(* CODESYS project TripleDoor.project

Project tree, tasks and I/O mapping:
  Device : CODESYS Control Win V3 x64, 3S - Smart Software Solutions GmbH, version 3.5.11.0
    application Application
      libraries: Standard, * (System); VisuDialogs, * (System); Util, * (System)
      task MainTask (cyclic, interval t#10ms, priority 1) calls Plant, Controller
      program Plant [ST]
      visualisation Visualization
      global variables GVL
      program Controller [ST]
  text list GlobalTextList
*)

// Device/Application/GVL
{attribute 'qualified_only' := 'false'}
VAR_GLOBAL
    (* Presence sensors *)
    presenceSideA           : BOOL;
    presenceSideB           : BOOL;
    (* Presence triggers - visualization writes here *)
    presenceTriggerA        : BOOL;
    presenceTriggerB        : BOOL;
    (* Partition pressure sensor *)
    partitionPressure       : BOOL;
    (* Manual rotation buttons *)
    rotateForwardButton     : BOOL;
    rotateBackwardButton    : BOOL;
    (* Rotation direction: FALSE=counter-clockwise (default), TRUE=clockwise *)
    rotationClockwise       : BOOL;
    (* Door angle sensor *)
    doorAngle               : REAL;
(* Rotation status *)
    isRotating              : BOOL;
    (* Motor control *)
    motorOn                 : BOOL;
    rotationForward         : BOOL;
    (* Motor enable switch *)
    motorEnable             : BOOL := TRUE;
    (* Emergency stop *)
    emergencyStop           : BOOL;
    (* Traffic lights *)
    lightSideA              : BOOL;
    lightSideB              : BOOL;
END_VAR

// Device/Application/Plant
PROGRAM Plant
VAR CONSTANT
    ROTATION_SPEED  : REAL := 0.1;
    MAX_ANGLE       : REAL := 360.0;
    PRESENCE_HOLD   : INT := 500;
END_VAR
VAR
    initialized      : BOOL := FALSE;
    presenceTimerA   : INT := 0;
    presenceTimerB   : INT := 0;
END_VAR

IF NOT initialized THEN
    GVL.doorAngle            := 0.0;
    GVL.presenceSideA        := FALSE;
    GVL.presenceSideB        := FALSE;
    GVL.presenceTriggerA     := FALSE;
    GVL.presenceTriggerB     := FALSE;
    presenceTimerA           := 0;
    presenceTimerB           := 0;
    initialized              := TRUE;
END_IF

(* Presence hold - trigger is set by visualization, timer keeps presence active *)
IF GVL.presenceTriggerA THEN
    presenceTimerA := PRESENCE_HOLD;
    GVL.presenceTriggerA := FALSE;
END_IF
GVL.presenceSideA := (presenceTimerA > 0);
IF presenceTimerA > 0 THEN
    presenceTimerA := presenceTimerA - 1;
END_IF

IF GVL.presenceTriggerB THEN
    presenceTimerB := PRESENCE_HOLD;
    GVL.presenceTriggerB := FALSE;
END_IF
GVL.presenceSideB := (presenceTimerB > 0);
IF presenceTimerB > 0 THEN
    presenceTimerB := presenceTimerB - 1;
END_IF

(* MotorSim *)
GVL.isRotating := GVL.motorOn;

(* DoorRotationSim *)
IF GVL.isRotating THEN
    IF GVL.rotationForward THEN
        GVL.doorAngle := GVL.doorAngle - ROTATION_SPEED;
    ELSE
        GVL.doorAngle := GVL.doorAngle + ROTATION_SPEED;
    END_IF
END_IF

IF GVL.doorAngle >= MAX_ANGLE THEN
    GVL.doorAngle := GVL.doorAngle - MAX_ANGLE;
END_IF
IF GVL.doorAngle < 0.0 THEN
    GVL.doorAngle := GVL.doorAngle + MAX_ANGLE;
END_IF

END_PROGRAM

// Device/Application/Controller
PROGRAM Controller
VAR CONSTANT
    ROTATION_TIME   : INT := 100;
    REVERSE_TICKS   : INT := 50;    (* 5 degrees at ROTATION_SPEED=0.1 *)
END_VAR
VAR
    (* MainControl state: 0=idle, 1=rotating, 2=manualRotation, 3=pressure *)
    mainState               : INT := 0;
    timer                   : INT := 0;
    manualActive            : BOOL := FALSE;
    manualDirectionForward  : BOOL := TRUE;
    (* Pressure sub-process: 0=released, 1=reversing, 2=stopped *)
    pauseState              : INT := 0;
    reverseCounter          : INT := 0;
END_VAR

(* Emergency stop - disable motor *)
IF GVL.emergencyStop THEN
    GVL.motorEnable := FALSE;
END_IF

(* Motor disabled - immediate stop, reset to idle *)
IF NOT GVL.motorEnable THEN
    GVL.motorOn := FALSE;
    GVL.rotationForward := NOT GVL.rotationClockwise;
    GVL.lightSideA := FALSE;
    GVL.lightSideB := FALSE;
	GVL.presenceSideA := FALSE;	
    GVL.presenceSideB := FALSE;
    manualActive := FALSE;
    timer := 0;
    pauseState := 0;
    mainState := 0;
ELSE

CASE mainState OF

0: (* idle *)
    GVL.lightSideA := TRUE;
    GVL.lightSideB := TRUE;
    IF GVL.rotateForwardButton AND NOT GVL.rotateBackwardButton AND NOT GVL.partitionPressure THEN
        manualActive := TRUE;
        manualDirectionForward := TRUE;
        GVL.motorOn := TRUE;
        GVL.rotationForward := NOT GVL.rotationClockwise;
        GVL.lightSideA := TRUE;
        GVL.lightSideB := TRUE;
        mainState := 2;

    ELSIF GVL.rotateBackwardButton AND NOT GVL.rotateForwardButton AND NOT GVL.partitionPressure THEN
        manualActive := TRUE;
        manualDirectionForward := FALSE;
        GVL.motorOn := TRUE;
        GVL.rotationForward := GVL.rotationClockwise;
        GVL.lightSideA := TRUE;
        GVL.lightSideB := TRUE;
        mainState := 2;

    ELSIF (GVL.presenceSideA OR GVL.presenceSideB) AND NOT GVL.partitionPressure THEN
        manualActive := FALSE;
        manualDirectionForward := TRUE;
        GVL.motorOn := TRUE;
        GVL.rotationForward := NOT GVL.rotationClockwise;
        GVL.lightSideA := TRUE;
        GVL.lightSideB := TRUE;
        timer := ROTATION_TIME;
        mainState := 1;
    END_IF

1: (* rotating *)
    IF (GVL.presenceSideA OR GVL.presenceSideB) THEN
        timer := ROTATION_TIME;
    END_IF

    IF GVL.partitionPressure THEN
        GVL.motorOn := FALSE;
        GVL.rotationForward := NOT GVL.rotationForward;
        GVL.lightSideA := FALSE;
        GVL.lightSideB := FALSE;
        reverseCounter := REVERSE_TICKS;
        pauseState := 1;
        mainState := 3;
    END_IF

    IF mainState = 1 THEN
        timer := timer - 1;
    END_IF
    IF timer <= 0 AND mainState = 1 THEN
        GVL.motorOn := FALSE;
        GVL.rotationForward := NOT GVL.rotationClockwise;
        GVL.lightSideA := TRUE;
        GVL.lightSideB := TRUE;
        mainState := 0;
    END_IF

2: (* manualRotation *)
    IF GVL.partitionPressure THEN
        GVL.motorOn := FALSE;
        GVL.rotationForward := NOT GVL.rotationForward;
        GVL.lightSideA := FALSE;
        GVL.lightSideB := FALSE;
        reverseCounter := REVERSE_TICKS;
        pauseState := 1;
        mainState := 3;

    ELSIF GVL.rotateForwardButton AND GVL.rotateBackwardButton THEN
        GVL.motorOn := FALSE;
        GVL.rotationForward := NOT GVL.rotationClockwise;
        GVL.lightSideA := TRUE;
        GVL.lightSideB := TRUE;
        manualActive := FALSE;
        mainState := 0;

    ELSIF manualDirectionForward AND GVL.rotateForwardButton THEN
        GVL.motorOn := TRUE;
        GVL.rotationForward := NOT GVL.rotationClockwise;
        GVL.lightSideA := TRUE;
        GVL.lightSideB := TRUE;

    ELSIF (NOT manualDirectionForward) AND GVL.rotateBackwardButton THEN
        GVL.motorOn := TRUE;
        GVL.rotationForward := GVL.rotationClockwise;
        GVL.lightSideA := TRUE;
        GVL.lightSideB := TRUE;

    ELSE
        GVL.motorOn := FALSE;
        GVL.rotationForward := NOT GVL.rotationClockwise;
        GVL.lightSideA := TRUE;
        GVL.lightSideB := TRUE;
        manualActive := FALSE;
        mainState := 0;
    END_IF

3: (* pressure reaction *)
    IF pauseState = 1 THEN
        (* Reversing 5 degrees *)
        GVL.motorOn := TRUE;
        reverseCounter := reverseCounter - 1;
        IF reverseCounter <= 0 THEN
            GVL.motorOn := FALSE;
            pauseState := 2;
        END_IF
    END_IF

    IF pauseState = 2 THEN
        (* Stopped until pressure released *)
        GVL.motorOn := FALSE;
        IF NOT GVL.partitionPressure THEN
            pauseState := 0;
        END_IF
    END_IF

    IF pauseState = 0 THEN
        (* Pressure released - resume *)
        IF manualActive THEN
            IF manualDirectionForward AND GVL.rotateForwardButton THEN
                GVL.motorOn := TRUE;
                GVL.rotationForward := NOT GVL.rotationClockwise;
                GVL.lightSideA := TRUE;
                GVL.lightSideB := TRUE;
                mainState := 2;
            ELSIF (NOT manualDirectionForward) AND GVL.rotateBackwardButton THEN
                GVL.motorOn := TRUE;
                GVL.rotationForward := GVL.rotationClockwise;
                GVL.lightSideA := TRUE;
                GVL.lightSideB := TRUE;
                mainState := 2;
            ELSE
                GVL.motorOn := FALSE;
                GVL.rotationForward := NOT GVL.rotationClockwise;
                GVL.lightSideA := TRUE;
                GVL.lightSideB := TRUE;
                manualActive := FALSE;
                mainState := 0;
            END_IF
        ELSIF timer > 0 THEN
            GVL.motorOn := TRUE;
            GVL.rotationForward := NOT GVL.rotationClockwise;
            GVL.lightSideA := TRUE;
            GVL.lightSideB := TRUE;
            mainState := 1;
        ELSE
            GVL.motorOn := FALSE;
            GVL.rotationForward := NOT GVL.rotationClockwise;
            GVL.lightSideA := TRUE;
            GVL.lightSideB := TRUE;
            mainState := 0;
        END_IF
    END_IF

END_CASE

END_IF (* motorEnable / emergencyStop *)

END_PROGRAM

// Device/Application/Visualization
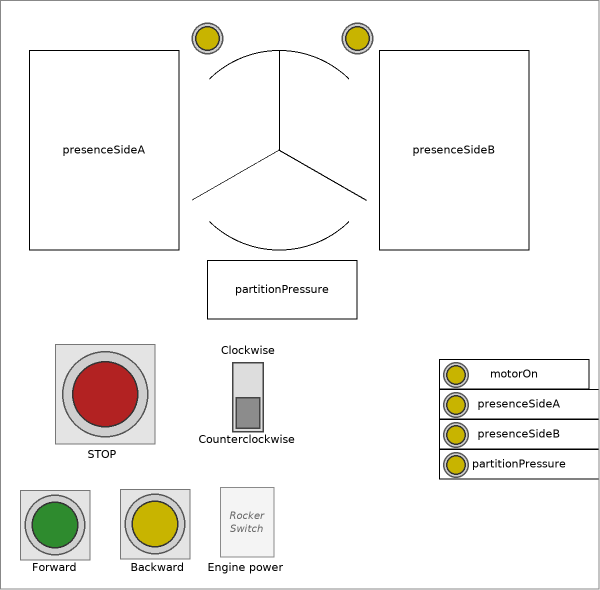
VISUALIZATION Visualization  // 600x590
    Rectangle (52,429 100x51), "STOP"
    Ellipse (179,50 200x200)
    Rectangle (59,50 150x200)
    Rectangle (349,50 150x200)
    RoundedRectangle (29,50 150x200), "presenceSideA"
        OnMouseMove: execute { GVL.presenceTriggerA := TRUE; }
        OnMouseEnter: execute { GVL.presenceTriggerA := TRUE; }
    RoundedRectangle (379,50 150x200), "presenceSideB"
        OnMouseMove: execute { GVL.presenceTriggerB := TRUE; }
        OnMouseEnter: execute { GVL.presenceTriggerB := TRUE; }
    PushSwitch (51,344 108x100), tooltip "Backward", variable: GVL.emergencyStop, behaviour: TAP, style: Switch-PushSwitch-Red
    Lamp1 (339,20 37x37), variable: GVL.lightSideB, style: Lamp-Lamp1-Yellow
    Lamp1 (189,20 37x37), variable: GVL.lightSideA, style: Lamp-Lamp1-Yellow
    Polyline (279,50) (279,150) (366,200) (279,150) (192,200)
        p2858320360: GVL.doorAngle
    Rectangle (207,260 150x59), "partitionPressure"
        OnMouseLeave: execute { GVL.partitionPressure := FALSE; }
        OnMouseEnter: execute { GVL.partitionPressure := TRUE; }
    Group (439,359 160x31)
        RoundedRectangle (0,0 150x30), "motorOn"
        Lamp1 (2,1 30x30), variable: GVL.motorOn, style: Lamp-Lamp1-Yellow
    RoundedRectangle (439,389 160x30), "presenceSideA"
    Lamp1 (441,390 30x30), variable: GVL.presenceSideA, style: Lamp-Lamp1-Yellow
    RoundedRectangle (439,419 160x30), "presenceSideB"
    Lamp1 (441,420 30x30), variable: GVL.presenceSideB, style: Lamp-Lamp1-Yellow
    RoundedRectangle (439,449 160x30), "partitionPressure"
    Lamp1 (441,450 30x30), variable: GVL.partitionPressure, style: Lamp-Lamp1-Yellow
    Rectangle (10,553 89x29), "Forward"
    Rectangle (113,553 89x29), "Backward"
    Rectangle (201,553 89x29), "Engine power"
    RockerSwitch (220,487 54x70), tooltip "Engine", variable: GVL.motorEnable, behaviour: TOGGLE, style: Switch-RockerSwitch-Red
    PushSwitch (120,489 70x70), tooltip "Backward", variable: GVL.rotateBackwardButton, behaviour: TAP, style: Switch-PushSwitch-Yellow
    PushSwitch (20,490 70x70), tooltip "Forward", variable: GVL.rotateForwardButton, behaviour: TAP, style: Switch-PushSwitch-Green
    Rectangle (192,425 110x29), "Counterclockwise"
    Rectangle (193,336 110x29), "Clockwise"
    DipSwitch (213,362 70x70), variable: GVL.rotationClockwise, behaviour: TOGGLE, style: Switch-DipSwitch-Gray
END_VISUALIZATION
